(*
Nazwa:			E_LidFeederState
Opis:			Stan zpodajnika platynek
Wersja:			v0.2
Data:			2018-10-18
Autor:			TW
Urzadzenia:		
Konfiguracja:	
Info:
*)

TYPE E_LidFeederState :
(
	eDisabled:=0,	//Wyłączona
	eError:=1,		//Błąd
	eManualMovement:=2,	//Tryb serwisowy
	eHoming:=3,		//Bazowanie
	eHomingDone:=4,	//Koniec bazowania
	eHeaterNotReady:=5,	//Grzanie
	eReady:=6,		//Gotowość
	eSuckingLid:=7,	//Pobieranie
	ePuttingLid:=8,	//Przygotowanie do odlożenia
	ePuttingLid2:=9,	//Nakładanie ostatnie
	eHeating:=10,	//Zgrzewanie
	eLidPutted:=11,	//Odłożona
	eGoingUp:=12,	//Podnoszenie
	ePreparingToDisable:=13 (*NOWY*) //Przygotowanie do wyłączenia
(**)
):=eDisabled;
END_TYPE

(* stored: Version 1.1.0.1, ProductVersion 3.1.4026.13, FileIdentifier 988f45aff3b5c92f88a5f2faae9ad7be51ec9795, FileSignature 24d7088a4e52db22c7c42a5de4a4769e9fb8fd0937c1991a89e27920eda0117f5ddc11a2b768be4ffcbd8ca28320cb692601dcbaa67369cc8fb286fb08c475243a07a2d50c7b084ddb4667fb7c8cc470447727c22eefdf647e9a702df5b5f99bf9659d08fdaf0af5e9348bee4cbf823c0465fc153f6c23a9b97a620ff2e5c5ba62ae0e20c5bb7dfc19acd48423c01dfd1d165c8a8b979841d3705b4279eb4b666acf51307019296d0e5cecd04aeeaaa2b198cb3a29608192bed76041edc3d129090cad26fd8597f0233104e5d45a0237bb00f2487bfde445edc875716d5fd25f61ad25d93ebed93308c82154b3e6a64d4753d099ad0a77afb7a53bfab82f1d33
   DUT E_LidFeederState: Id {64ecfeb0-78d5-4891-a519-98cde606399d} *)
